// TIA Portal V17 export
// export: Created 2025-04-11T04:54:23.7235902Z, ExportSetting WithDefaults, DisplayName Totally Integrated Automation Portal, DisplayVersion V17, DisplayName TIA Portal Openness, DisplayVersion V17, DisplayName TIA Portal Version Control Interface, DisplayVersion V17, DisplayName SINAMICS Startdrive Advanced, DisplayVersion V17, DisplayName SINAMICS Startdrive G130, G150, S120, S150, SINAMICS MV, S210, DisplayVersion V17, DisplayName SINAMICS Startdrive G110M, G120, G120C, G120D, G120P, G115D, DisplayVersion V17, DisplayName STEP 7 Professional, DisplayVersion V17, DisplayName STEP 7 Safety, DisplayVersion V17, DisplayName WinCC Advanced, DisplayVersion V17
TYPE "UDT_Valve_HMI"
// stored: IsFailsafeCompliant false
   STRUCT
      IN_xNormOpen : Bool;   // 常开常闭阀选择/常开为1，常闭为0
      IN_xManualOpen : Bool;   // 手动开
      IN_xManualClose : Bool;   // 手动关
      IN_xCounterReset : Bool;   // 计数复位
      OUT_uiState : UInt;   // 状态字(0=初始状态,1=已关闭,2=已打开,3=正在打开,4=正在关闭,5=关阀故障,6=开阀故障,7=传感器故障)
   END_STRUCT;
END_TYPE
